FUNCTION Convert_BOOL_TO_DATE : BOOL
VAR_INPUT
	in : BOOL;
	out : REFERENCE TO DATE;
END_VAR

out := BOOL_TO_DATE(in);
Convert_BOOL_TO_DATE := TRUE;

END_FUNCTION

(* stored: Version 1.1.0.1, ProductVersion 3.1.4024.12
   POU Convert_BOOL_TO_DATE: Id {9046aacb-54d7-443b-8c42-1fda59e16ca1}, SpecialFunc None *)
